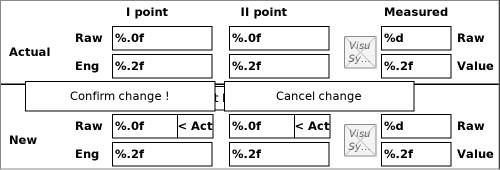
VISUALIZATION MeasureCalibration_NoTitle  // 500x170
VAR_IN_OUT
	stMeasureData:stMeasurementScalingData;
END_VAR
VAR_INPUT
	diAnalogIn:DINT;
END_VAR
VAR
	rRaw1:REAL;
	rRaw2:REAL:= 32767;
	rEng1:REAL;
	rEng2:REAL;
	bConfirmation:BOOL:=FALSE;
END_VAR
    Rectangle (0,0 500x84)
    Rectangle (112,26 100x24), "%.0f", text variable: stMeasureData.rScalingRawValue_I, input disabled if: TRUE
    Label (72,26 40x24), "Raw"
    Rectangle (112,54 100x24), "%.2f", text variable: stMeasureData.rScalingEngValue_I, input disabled if: TRUE
    Label (72,54 40x24), "Eng"
    Label (112,0 70x24), "I point"
    Rectangle (229,26 100x24), "%.0f", text variable: stMeasureData.rScalingRawValue_II, input disabled if: TRUE
    Rectangle (229,54 100x24), "%.2f", text variable: stMeasureData.rScalingEngValue_II, input disabled if: TRUE
    Label (229,0 70x24), "II point"
    Image (344,36 32x32), image: VisuSymbols.Symbols.ArrowBoldRight
    Label (381,0 70x24), "Measured"
    Rectangle (381,54 70x24), "%.2f", text variable: ( (DINT_TO_REAL(diAnalogIn) - stMeasureData.rScalingRawValue_I)/ ( LIMIT(0.1,(stMeasureData.rScalingRawValue_II - stMeasureData.rScalingRawValue_I),999999999999)))*( stMeasureData.rScalingEngValue_II - stMeasureData.rScalingEngValue_I)+stMeasureData.rScalingEngValue_I, input disabled if: TRUE
    Rectangle (381,26 70x24), "%d", text variable: diAnalogIn, input disabled if: TRUE
    Label (454,26 40x24), "Raw"
    Label (454,54 40x24), "Value"
    Rectangle (0,84 500x85)
    Rectangle (112,114 68x24), "%.0f", text variable: rRaw1
        OnMouseClick: write rRaw1 via Default, title 'New Raw I value', format %.0f
    Label (72,114 40x24), "Raw"
    Rectangle (112,142 100x24), "%.2f", text variable: rEng1
        OnMouseClick: write rEng1 via Default, title 'New Eng I value', format %.2f
    Label (72,142 40x24), "Eng"
    Rectangle (229,114 68x24), "%.0f", text variable: rRaw2
        OnMouseClick: write rRaw2 via Default, title 'New Raw II value', format %.0f
    Rectangle (229,142 100x24), "%.2f", text variable: rEng2
        OnMouseClick: write rEng2 via Default, title 'New Eng II value', format %.2f
    Image (344,124 32x32), image: VisuSymbols.Symbols.ArrowBoldRight
    Rectangle (381,142 70x24), "%.2f", text variable: ( (DINT_TO_REAL(diAnalogIn) - rRaw1)/ (LIMIT(1,(rRaw2 - rRaw1),9999999999999) ) ) * ( rEng2 - rEng1)+ rEng1, input disabled if: TRUE
    Rectangle (381,114 70x24), "%d", text variable: diAnalogIn, input disabled if: TRUE
    Label (454,114 40x24), "Raw"
    Label (454,142 40x24), "Value"
    Label (6,128 40x24), "New"
    Label (6,40 40x24), "Actual"
    RoundedRectangle (113,86 216x24), "/\ /\ /\ Set NEW /\ /\ /\", invisible if: bConfirmation
        toggle bConfirmation
    RoundedRectangle (177,114 36x24), "< Act"
        OnMouseClick: execute { rRaw1:= DINT_TO_REAL(diAnalogIn); }
    RoundedRectangle (294,114 36x24), "< Act"
        OnMouseClick: execute { rRaw2 := DINT_TO_REAL(diAnalogIn); }
    RoundedRectangle (25,81 190x30), "Confirm change !", invisible if: NOT bConfirmation
        OnMouseClick: execute {
            stMeasureData.rScalingEngValue_I := rEng1;
            stMeasureData.rScalingEngValue_II := rEng2;
            stMeasureData.rScalingRawValue_I := rRaw1;
            stMeasureData.rScalingRawValue_II := rRaw2;
            bConfirmation:= FALSE;
        }
    RoundedRectangle (224,81 190x30), "Cancel change", invisible if: NOT bConfirmation
        OnMouseClick: execute { bConfirmation:= FALSE; }
END_VISUALIZATION

(* stored: Version 1.1.0.1, ProductVersion 3.1.4024.12
   Visu MeasureCalibration_NoTitle: Id {dcb201f9-e7ef-48ab-aefa-484dc47f3847} *)
